TYPE Figure :
STRUCT
	length : INT := 0;
    X : ARRAY[0..9999] OF REAL := [10000(0)];
    Y : ARRAY[0..9999] OF REAL := [10000(0)];
	Visu : ARRAY[0..200] OF VisuElems.VisuStructPoint;
END_STRUCT
END_TYPE

(* stored: Version 1.1.0.1, ProductVersion 3.1.4024.12
   DUT Figure: Id {eca3ee30-3f47-4b1f-9248-b3b7311b65a7} *)
